(* IEC 61131-3 sources: HappyLearnCodesys/content/softmotion/CNC06_File_3DPath, 3 files *)

(* ---- GVL.st ---- *)
VAR_GLOBAL CONSTANT
	gc_dwCycle : DWORD := 4000;
END_VAR

(* ---- CNC.st ---- *)
PROGRAM CNC
VAR
	iState: INT;
	pX, pY, pZ: MC_Power;

	ipo: SMC_Interpolator;
	trafo: SMC_TRAFO_Gantry3;
	trafof: SMC_TRAFOF_Gantry3D;
	cabpX, 	cabpY, 	cabpZ: SMC_ControlAxisByPos;

	pt: SMC_PositionTracker;
	pointbuffer_pt: ARRAY [0..1000] OF VisuStruct3DPathPoint;

END_VAR

pX(
	Enable:=TRUE ,
	bRegulatorOn:=TRUE ,
	bDriveStart:=TRUE ,
	Axis:=AxisX);
pY(
	Enable:=TRUE ,
	bRegulatorOn:=TRUE ,
	bDriveStart:=TRUE ,
	Axis:=AxisY);
pZ(
	Enable:=TRUE ,
	bRegulatorOn:=TRUE ,
	bDriveStart:=TRUE ,
	Axis:=AxisZ);

CASE iState OF
0:
	IF pX.Status AND pY.Status AND pZ.Status THEN
		iState:=100;
	END_IF
100:
	Interpolation();
END_CASE

(* ---- CNC_PreparePath.st ---- *)
PROGRAM CNC_PreparePath
VAR_INPUT
	xStart: BOOL;
	sFileName: STRING := '_cnc/CNC1.cnc';
END_VAR
VAR_OUTPUT
	xStartIpo: BOOL;
	poqPath: Pointer to SMC_Outqueue;
END_VAR
VAR
	iState: INT;
	rncf2 : SMC_ReadNCFile2;
	nci: SMC_NCInterpreter;
	cv: SMC_CheckVelocities;
	agiBufInterpreter: ARRAY[0..99] OF SMC_GeoInfo;

	pcf: SMC_PathCopierFile;
	pointbuffer: ARRAY [0..1000] OF VisuStruct3DPathPoint;

	vc: VisuStruct3DControl;
END_VAR

poqPath := cv.poqDataOut;

CASE iState OF
0:	// idle
	IF xStart THEN
		iState := 10;
		xStartIpo := FALSE;
		rncf2(bExecute:= FALSE);
		nci(bExecute:= FALSE, sentences:= rncf2.sentences);
		cv(bExecute:= FALSE);

		pcf(bExecute:= FALSE ,
			udiNumberOfPointsInArray:= SIZEOF(pointbuffer)/SIZEOF(pointbuffer[0]) ,
			pBuffer:= ADR(pointbuffer) ,
			sFileName:= sFilename);

		WHILE NOT (pcf.bDone OR pcf.bError) DO
			pcf(bExecute:= TRUE);
		END_WHILE

		xStart := FALSE;
	END_IF
10:	// start reading and processing
	rncf2(
		bExecute:= TRUE,
		sFileName:= sFilename);
	nci(
		bExecute:= TRUE,
		nSizeOutQueue:= SIZEOF(agiBufInterpreter),
		pbyBufferOutQueue:= ADR(agiBufInterpreter),
		sentences:= rncf2.sentences);
	cv(
		bExecute:= TRUE,
		poqDataIn:= nci.poqDataOut);

	xStartIpo := TRUE;
	IF NOT cv.bBusy THEN
		iState := 0;
	END_IF
END_CASE
